(* Logix 5000 project; controller Sucrose_Main Emulate 5570 rev 20.12; software revision 20.01; part 24 of 30 *)
(* tags used below, declared in another part *)
   AI_E23_0 : REAL[8];   // Analog Input EN2T_FLX 192.168.1.23
   AI_E23_1 : REAL[8];   // Analog Input EN2T_FLX 192.168.1.23
   Alarm_ACK_Master_Timer : TIMER;
   CIPRemote : Area_Program;
   DI_E23_3 : ALIAS FOR FLX_E23:3:I;   // Discrete Input EN2T_FLX 192.168.1.23
   DI_E23_4 : ALIAS FOR FLX_E23:4:I;   // Discrete Input EN2T_FLX 192.168.1.23
   DI_E25_2 : ALIAS FOR FLX_E25:2:I;   // Discrete Input EN2T_FLX 192.168.1.25
   DO_E24_0 : ALIAS FOR FLX_E24:0:O;   // Discrete Output EN2T_FLX 192.168.1.24
   DO_E24_1 : ALIAS FOR FLX_E24:1:O;   // Discrete Output EN2T_FLX 192.168.1.24
   FV230006_AOI : QSI_Flow_Valve;   // FV-23-00-06 RETURN PIG TO LAUNCHER VALVE V7
   FV230007_AOI : QSI_Flow_Valve;   // FV-23-00-07 RETURN PIG TO LAUNCHER VALVE V6
   FV230101_AOI : QSI_Flow_Valve;   // FV-23-01-01-O SUCROSE RECEIVING TO SUCROSE TANK #1 VALVE OPEN
   FV230201_AOI : QSI_Flow_Valve;   // FV-23-02-01-O SUCROSE RECEIVING TO SUCROSE TANK #2 VALVE OPEN
   FV230301_AOI : QSI_Flow_Valve;   // FV-23-03-01-O SUCROSE RECEIVING TO SUCROSE TANK #3 VALVE OPEN
   ONESHOTBITS : INT[10];
   Rung_Comment : BOOL;
   Sucrose_MM_Enable : BOOL;
   SucroseCIP_RECEIVING_REMOTE : CIP_REMOTE;
   SucroseCIP_TK230101_REMOTE : CIP_REMOTE;
   SucroseCIP_TK230201_REMOTE : CIP_REMOTE;
   SucroseCIP_TK230301_REMOTE : CIP_REMOTE;
   SucroseReceiving : Area_Program;
   SucroseTanks : Area_Program;
   TK_23_01_01_HIGH_LEVEL : DINT;
   TK_23_01_01_RECEIVING_COMPLETE : BOOL;
   TK_23_02_01_HIGH_LEVEL : DINT;
   TK_23_02_01_RECEIVING_COMPLETE : BOOL;
   TK_23_03_01_HIGH_LEVEL : DINT;
   TK_23_03_01_RECEIVING_COMPLETE : BOOL;
(* ReceivingArea_AutoLogic, continued *)

ROUTINE Enable_Logic   (* ladder *)
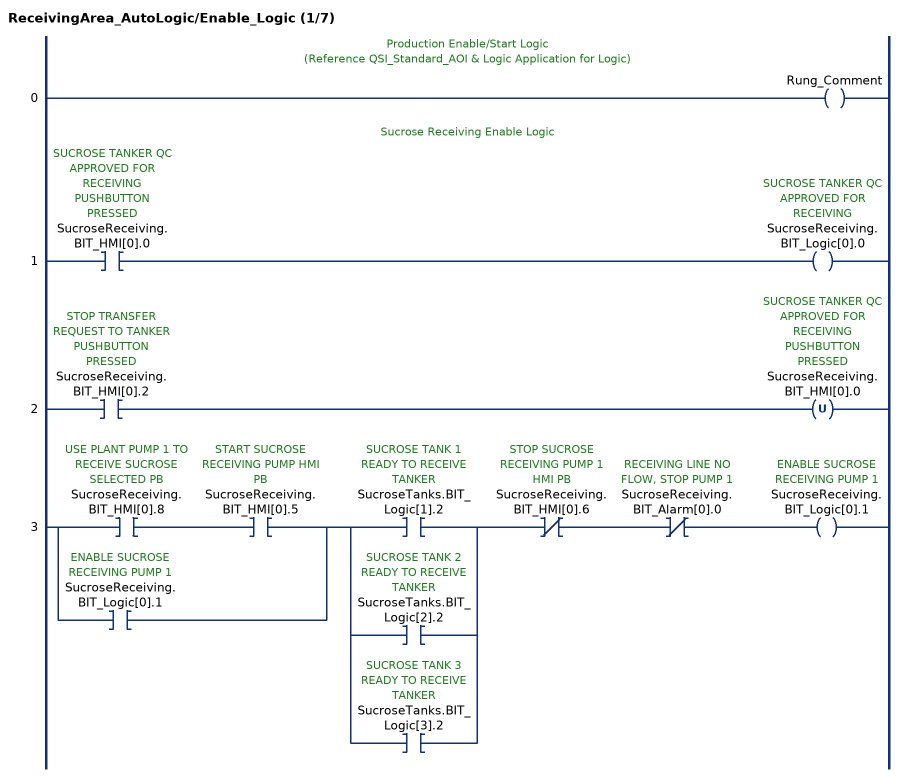
   // Production Enable/Start Logic
   // (Reference QSI_Standard_AOI & Logic Application for Logic)
   0: OTE(Rung_Comment);
   // Sucrose Receiving Enable Logic
   1: XIC(SucroseReceiving.BIT_HMI[0].0)OTE(SucroseReceiving.BIT_Logic[0].0);
   2: XIC(SucroseReceiving.BIT_HMI[0].2)OTU(SucroseReceiving.BIT_HMI[0].0);
   3: [XIC(SucroseReceiving.BIT_HMI[0].8) XIC(SucroseReceiving.BIT_HMI[0].5) ,XIC(SucroseReceiving.BIT_Logic[0].1) ][XIC(SucroseTanks.BIT_Logic[1].2) ,XIC(SucroseTanks.BIT_Logic[2].2) ,XIC(SucroseTanks.BIT_Logic[3].2) ]XIO(SucroseReceiving.BIT_HMI[0].6)XIO(SucroseReceiving.BIT_Alarm[0].0)OTE(SucroseReceiving.BIT_Logic[0].1);
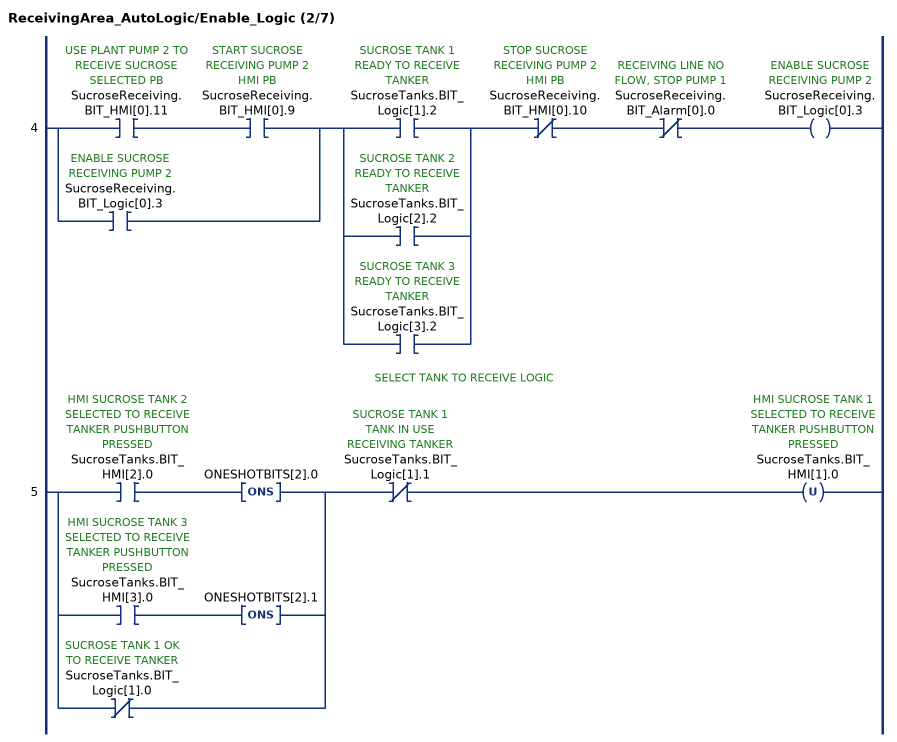
   4: [XIC(SucroseReceiving.BIT_HMI[0].11) XIC(SucroseReceiving.BIT_HMI[0].9) ,XIC(SucroseReceiving.BIT_Logic[0].3) ][XIC(SucroseTanks.BIT_Logic[1].2) ,XIC(SucroseTanks.BIT_Logic[2].2) ,XIC(SucroseTanks.BIT_Logic[3].2) ]XIO(SucroseReceiving.BIT_HMI[0].10)XIO(SucroseReceiving.BIT_Alarm[0].0)OTE(SucroseReceiving.BIT_Logic[0].3);
   // SELECT TANK TO RECEIVE LOGIC
   5: [XIC(SucroseTanks.BIT_HMI[2].0) ONS(ONESHOTBITS[2].0) ,XIC(SucroseTanks.BIT_HMI[3].0) ONS(ONESHOTBITS[2].1) ,XIO(SucroseTanks.BIT_Logic[1].0) ]XIO(SucroseTanks.BIT_Logic[1].1)OTU(SucroseTanks.BIT_HMI[1].0);
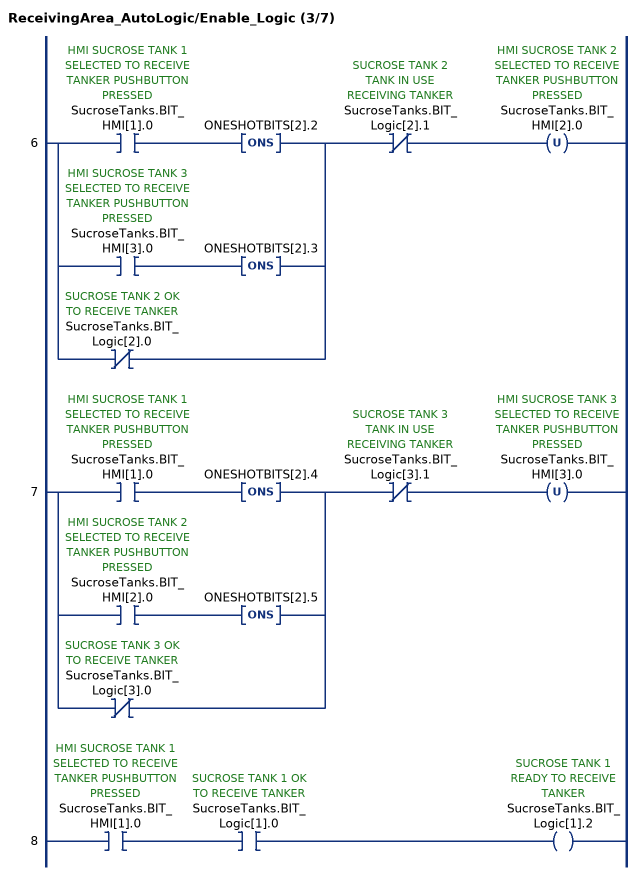
   6: [XIC(SucroseTanks.BIT_HMI[1].0) ONS(ONESHOTBITS[2].2) ,XIC(SucroseTanks.BIT_HMI[3].0) ONS(ONESHOTBITS[2].3) ,XIO(SucroseTanks.BIT_Logic[2].0) ]XIO(SucroseTanks.BIT_Logic[2].1)OTU(SucroseTanks.BIT_HMI[2].0);
   7: [XIC(SucroseTanks.BIT_HMI[1].0) ONS(ONESHOTBITS[2].4) ,XIC(SucroseTanks.BIT_HMI[2].0) ONS(ONESHOTBITS[2].5) ,XIO(SucroseTanks.BIT_Logic[3].0) ]XIO(SucroseTanks.BIT_Logic[3].1)OTU(SucroseTanks.BIT_HMI[3].0);
   8: XIC(SucroseTanks.BIT_HMI[1].0)XIC(SucroseTanks.BIT_Logic[1].0)OTE(SucroseTanks.BIT_Logic[1].2);
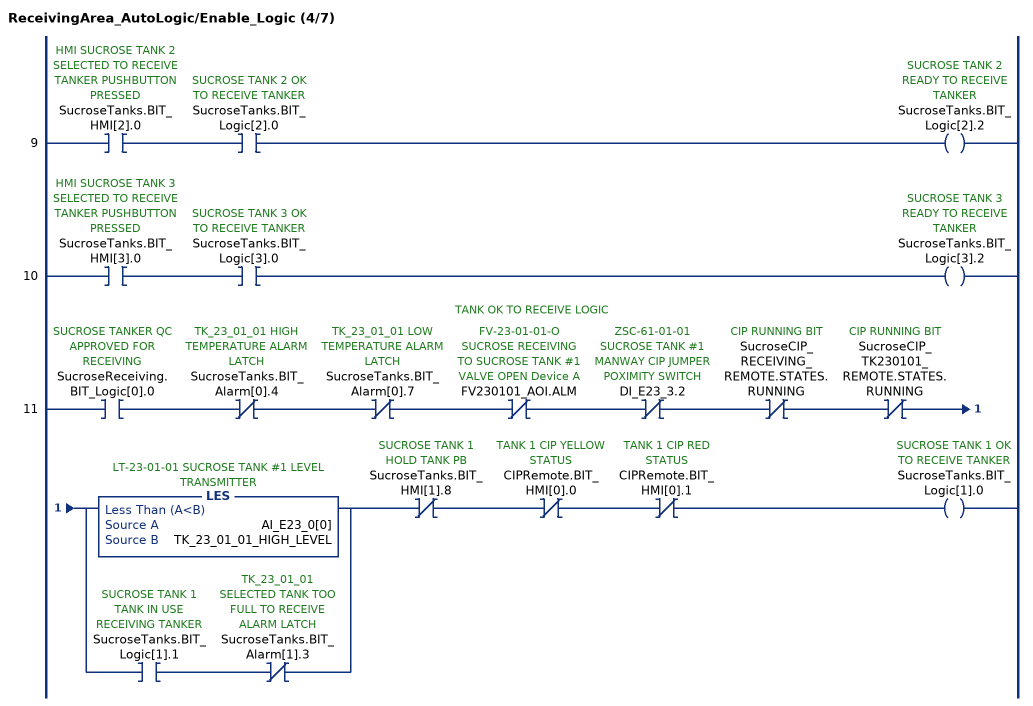
   9: XIC(SucroseTanks.BIT_HMI[2].0)XIC(SucroseTanks.BIT_Logic[2].0)OTE(SucroseTanks.BIT_Logic[2].2);
   10: XIC(SucroseTanks.BIT_HMI[3].0)XIC(SucroseTanks.BIT_Logic[3].0)OTE(SucroseTanks.BIT_Logic[3].2);
   // TANK OK TO RECEIVE LOGIC
   11: XIC(SucroseReceiving.BIT_Logic[0].0)XIO(SucroseTanks.BIT_Alarm[0].4)XIO(SucroseTanks.BIT_Alarm[0].7)XIO(FV230101_AOI.ALM)XIO(DI_E23_3.2)XIO(SucroseCIP_RECEIVING_REMOTE.STATES.RUNNING)XIO(SucroseCIP_TK230101_REMOTE.STATES.RUNNING)[LES(AI_E23_0[0],TK_23_01_01_HIGH_LEVEL) ,XIC(SucroseTanks.BIT_Logic[1].1) XIO(SucroseTanks.BIT_Alarm[1].3) ]XIO(SucroseTanks.BIT_HMI[1].8)XIO(CIPRemote.BIT_HMI[0].0)XIO(CIPRemote.BIT_HMI[0].1)OTE(SucroseTanks.BIT_Logic[1].0);
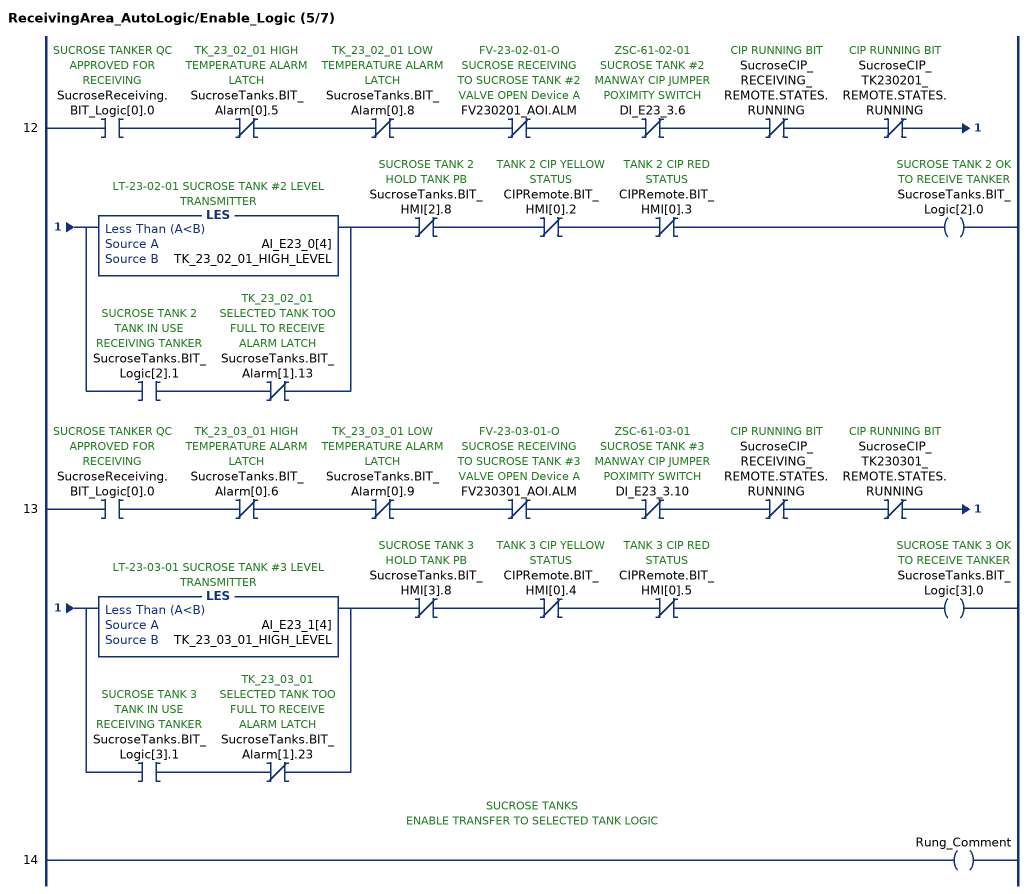
   12: XIC(SucroseReceiving.BIT_Logic[0].0)XIO(SucroseTanks.BIT_Alarm[0].5)XIO(SucroseTanks.BIT_Alarm[0].8)XIO(FV230201_AOI.ALM)XIO(DI_E23_3.6)XIO(SucroseCIP_RECEIVING_REMOTE.STATES.RUNNING)XIO(SucroseCIP_TK230201_REMOTE.STATES.RUNNING)[LES(AI_E23_0[4],TK_23_02_01_HIGH_LEVEL) ,XIC(SucroseTanks.BIT_Logic[2].1) XIO(SucroseTanks.BIT_Alarm[1].13) ]XIO(SucroseTanks.BIT_HMI[2].8)XIO(CIPRemote.BIT_HMI[0].2)XIO(CIPRemote.BIT_HMI[0].3)OTE(SucroseTanks.BIT_Logic[2].0);
   13: XIC(SucroseReceiving.BIT_Logic[0].0)XIO(SucroseTanks.BIT_Alarm[0].6)XIO(SucroseTanks.BIT_Alarm[0].9)XIO(FV230301_AOI.ALM)XIO(DI_E23_3.10)XIO(SucroseCIP_RECEIVING_REMOTE.STATES.RUNNING)XIO(SucroseCIP_TK230301_REMOTE.STATES.RUNNING)[LES(AI_E23_1[4],TK_23_03_01_HIGH_LEVEL) ,XIC(SucroseTanks.BIT_Logic[3].1) XIO(SucroseTanks.BIT_Alarm[1].23) ]XIO(SucroseTanks.BIT_HMI[3].8)XIO(CIPRemote.BIT_HMI[0].4)XIO(CIPRemote.BIT_HMI[0].5)OTE(SucroseTanks.BIT_Logic[3].0);
   // SUCROSE TANKS
   // ENABLE TRANSFER TO SELECTED TANK LOGIC
   14: OTE(Rung_Comment);
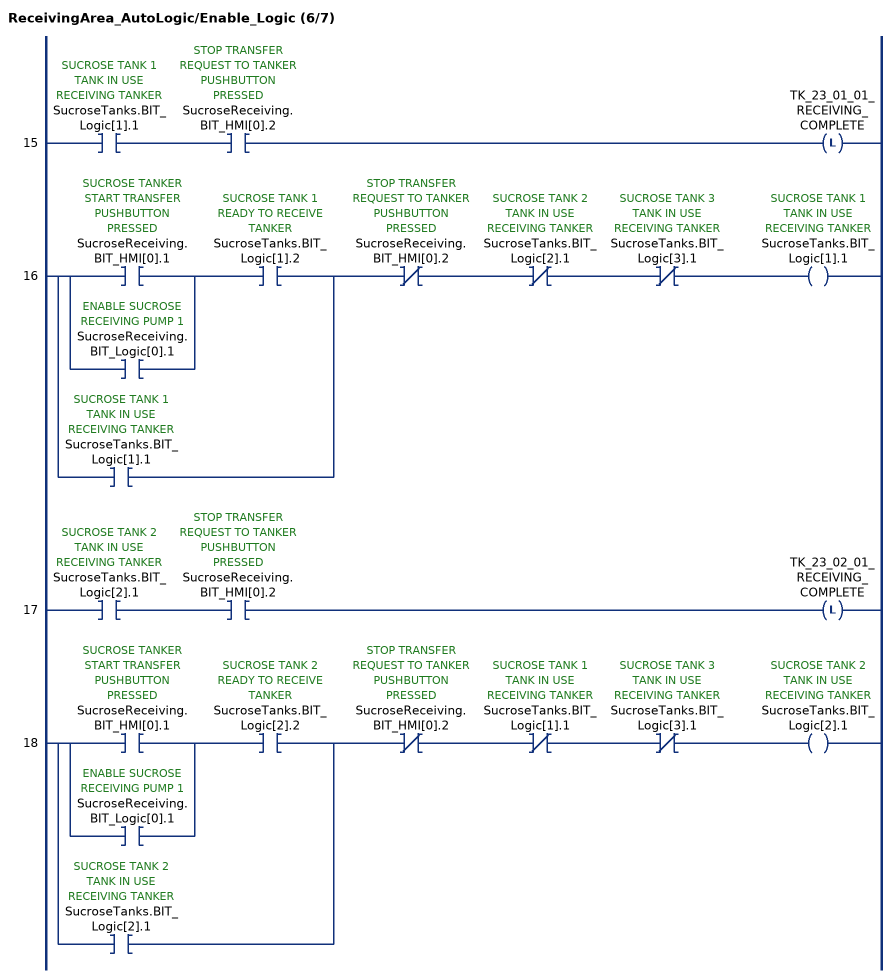
   15: XIC(SucroseTanks.BIT_Logic[1].1)XIC(SucroseReceiving.BIT_HMI[0].2)OTL(TK_23_01_01_RECEIVING_COMPLETE);
   16: [[XIC(SucroseReceiving.BIT_HMI[0].1) ,XIC(SucroseReceiving.BIT_Logic[0].1) ] XIC(SucroseTanks.BIT_Logic[1].2) ,XIC(SucroseTanks.BIT_Logic[1].1) ]XIO(SucroseReceiving.BIT_HMI[0].2)XIO(SucroseTanks.BIT_Logic[2].1)XIO(SucroseTanks.BIT_Logic[3].1)OTE(SucroseTanks.BIT_Logic[1].1);
   17: XIC(SucroseTanks.BIT_Logic[2].1)XIC(SucroseReceiving.BIT_HMI[0].2)OTL(TK_23_02_01_RECEIVING_COMPLETE);
   18: [[XIC(SucroseReceiving.BIT_HMI[0].1) ,XIC(SucroseReceiving.BIT_Logic[0].1) ] XIC(SucroseTanks.BIT_Logic[2].2) ,XIC(SucroseTanks.BIT_Logic[2].1) ]XIO(SucroseReceiving.BIT_HMI[0].2)XIO(SucroseTanks.BIT_Logic[1].1)XIO(SucroseTanks.BIT_Logic[3].1)OTE(SucroseTanks.BIT_Logic[2].1);
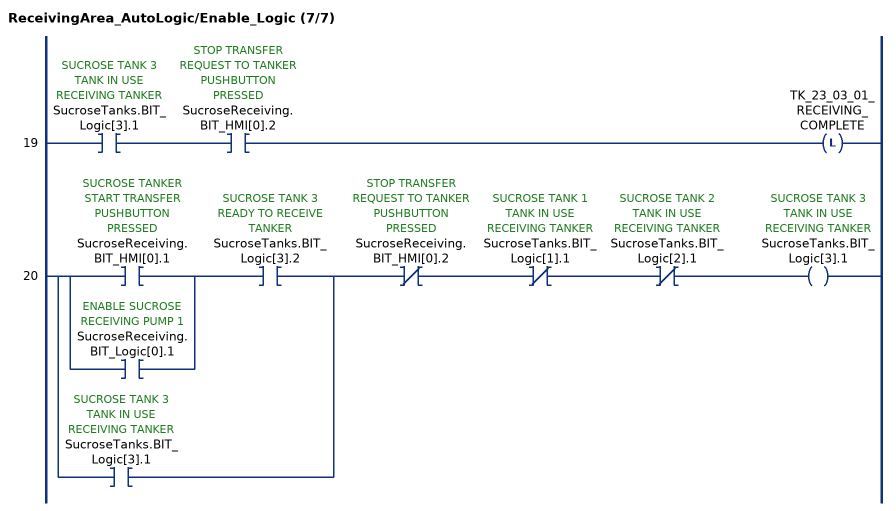
   19: XIC(SucroseTanks.BIT_Logic[3].1)XIC(SucroseReceiving.BIT_HMI[0].2)OTL(TK_23_03_01_RECEIVING_COMPLETE);
   20: [[XIC(SucroseReceiving.BIT_HMI[0].1) ,XIC(SucroseReceiving.BIT_Logic[0].1) ] XIC(SucroseTanks.BIT_Logic[3].2) ,XIC(SucroseTanks.BIT_Logic[3].1) ]XIO(SucroseReceiving.BIT_HMI[0].2)XIO(SucroseTanks.BIT_Logic[1].1)XIO(SucroseTanks.BIT_Logic[2].1)OTE(SucroseTanks.BIT_Logic[3].1);
END_ROUTINE

ROUTINE MainRoutine   (* ladder *)
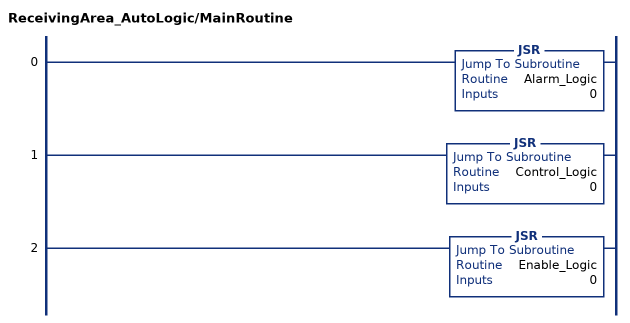
   0: JSR(Alarm_Logic,0);
   1: JSR(Control_Logic,0);
   2: JSR(Enable_Logic,0);
END_ROUTINE
END_PROGRAM

PROGRAM ReceivingArea_EN2T_IO_Discrete_DO_E24_0   (* main routine MainRoutine *)

ROUTINE _00_FV230006   (* ladder *)
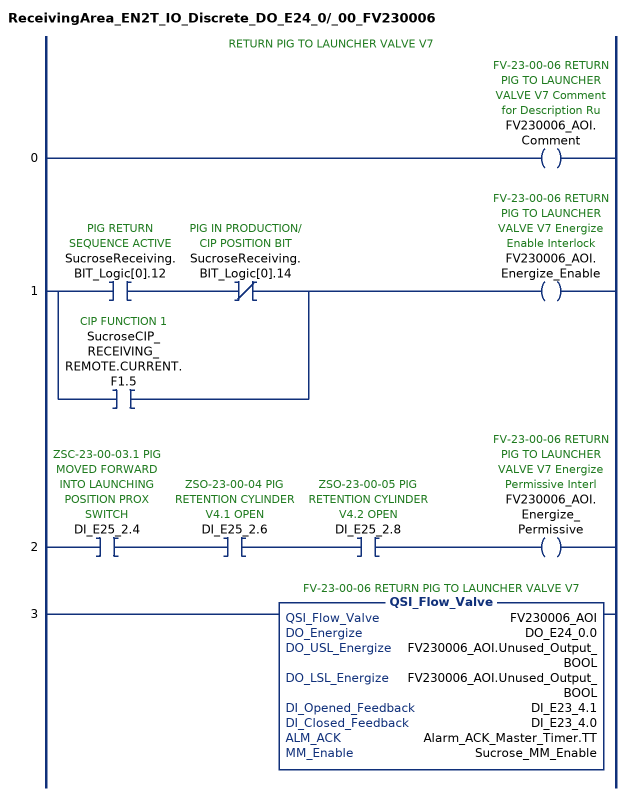
   // RETURN PIG TO LAUNCHER VALVE V7
   0: OTE(FV230006_AOI.Comment);
   1: [XIC(SucroseReceiving.BIT_Logic[0].12) XIO(SucroseReceiving.BIT_Logic[0].14) ,XIC(SucroseCIP_RECEIVING_REMOTE.CURRENT.F1.5) ]OTE(FV230006_AOI.Energize_Enable);
   2: XIC(DI_E25_2.4)XIC(DI_E25_2.6)XIC(DI_E25_2.8)OTE(FV230006_AOI.Energize_Permissive);
   3: QSI_Flow_Valve(FV230006_AOI,DO_E24_0.0,FV230006_AOI.Unused_Output_BOOL,FV230006_AOI.Unused_Output_BOOL,DI_E23_4.1,DI_E23_4.0,Alarm_ACK_Master_Timer.TT,Sucrose_MM_Enable);
END_ROUTINE

ROUTINE _01_FV230007   (* ladder *)
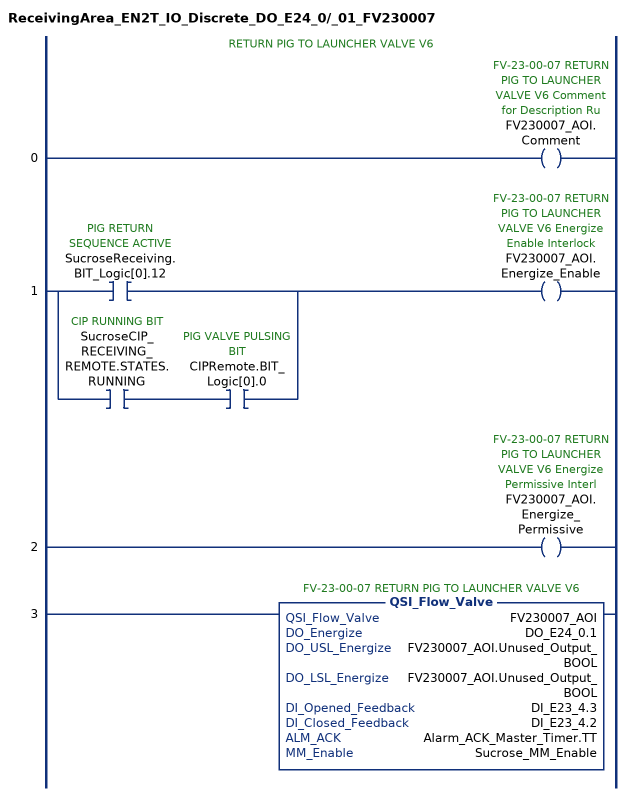
   // RETURN PIG TO LAUNCHER VALVE V6
   0: OTE(FV230007_AOI.Comment);
   1: [XIC(SucroseReceiving.BIT_Logic[0].12) ,XIC(SucroseCIP_RECEIVING_REMOTE.STATES.RUNNING) XIC(CIPRemote.BIT_Logic[0].0) ]OTE(FV230007_AOI.Energize_Enable);
   2: OTE(FV230007_AOI.Energize_Permissive);
   3: QSI_Flow_Valve(FV230007_AOI,DO_E24_0.1,FV230007_AOI.Unused_Output_BOOL,FV230007_AOI.Unused_Output_BOOL,DI_E23_4.3,DI_E23_4.2,Alarm_ACK_Master_Timer.TT,Sucrose_MM_Enable);
END_ROUTINE

ROUTINE _02_FV230101   (* ladder *)
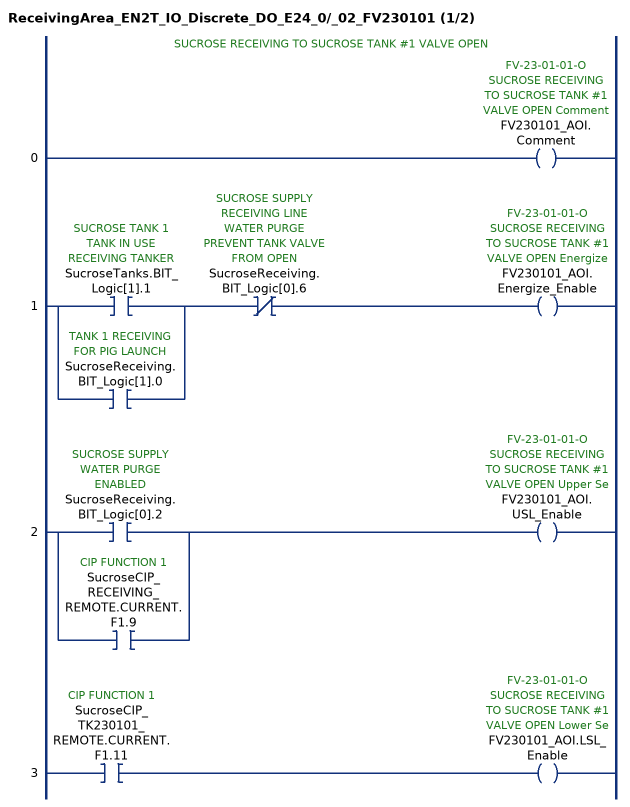
   // SUCROSE RECEIVING TO SUCROSE TANK #1 VALVE OPEN
   0: OTE(FV230101_AOI.Comment);
   1: [XIC(SucroseTanks.BIT_Logic[1].1) ,XIC(SucroseReceiving.BIT_Logic[1].0) ]XIO(SucroseReceiving.BIT_Logic[0].6)OTE(FV230101_AOI.Energize_Enable);
   2: [XIC(SucroseReceiving.BIT_Logic[0].2) ,XIC(SucroseCIP_RECEIVING_REMOTE.CURRENT.F1.9) ]OTE(FV230101_AOI.USL_Enable);
   3: XIC(SucroseCIP_TK230101_REMOTE.CURRENT.F1.11)OTE(FV230101_AOI.LSL_Enable);
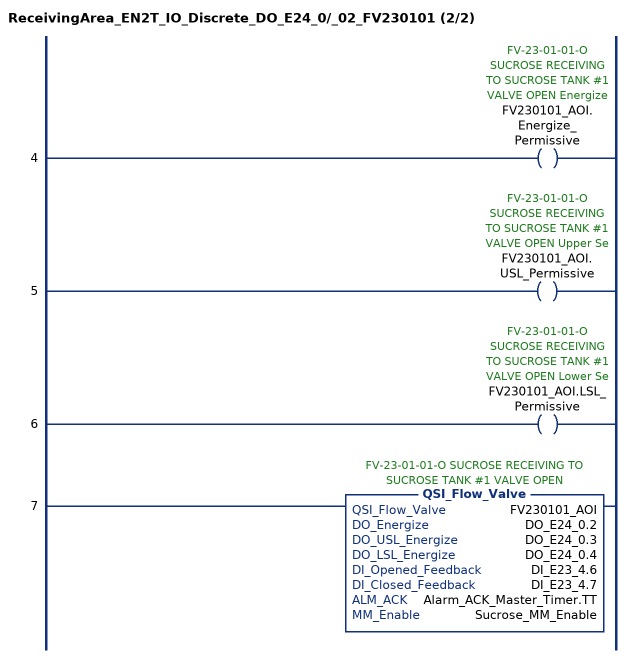
   4: OTE(FV230101_AOI.Energize_Permissive);
   5: OTE(FV230101_AOI.USL_Permissive);
   6: OTE(FV230101_AOI.LSL_Permissive);
   7: QSI_Flow_Valve(FV230101_AOI,DO_E24_0.2,DO_E24_0.3,DO_E24_0.4,DI_E23_4.6,DI_E23_4.7,Alarm_ACK_Master_Timer.TT,Sucrose_MM_Enable);
END_ROUTINE

ROUTINE _08_FV230201   (* ladder *)
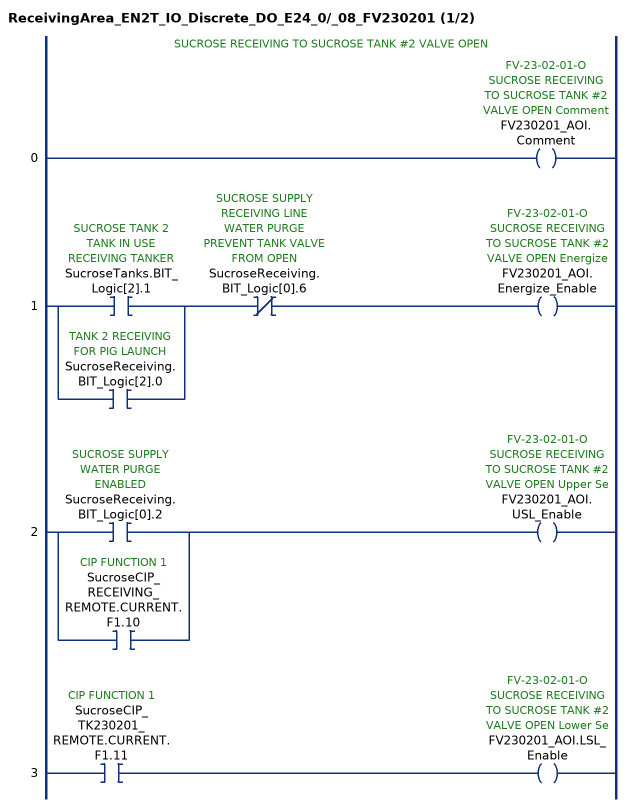
   // SUCROSE RECEIVING TO SUCROSE TANK #2 VALVE OPEN
   0: OTE(FV230201_AOI.Comment);
   1: [XIC(SucroseTanks.BIT_Logic[2].1) ,XIC(SucroseReceiving.BIT_Logic[2].0) ]XIO(SucroseReceiving.BIT_Logic[0].6)OTE(FV230201_AOI.Energize_Enable);
   2: [XIC(SucroseReceiving.BIT_Logic[0].2) ,XIC(SucroseCIP_RECEIVING_REMOTE.CURRENT.F1.10) ]OTE(FV230201_AOI.USL_Enable);
   3: XIC(SucroseCIP_TK230201_REMOTE.CURRENT.F1.11)OTE(FV230201_AOI.LSL_Enable);
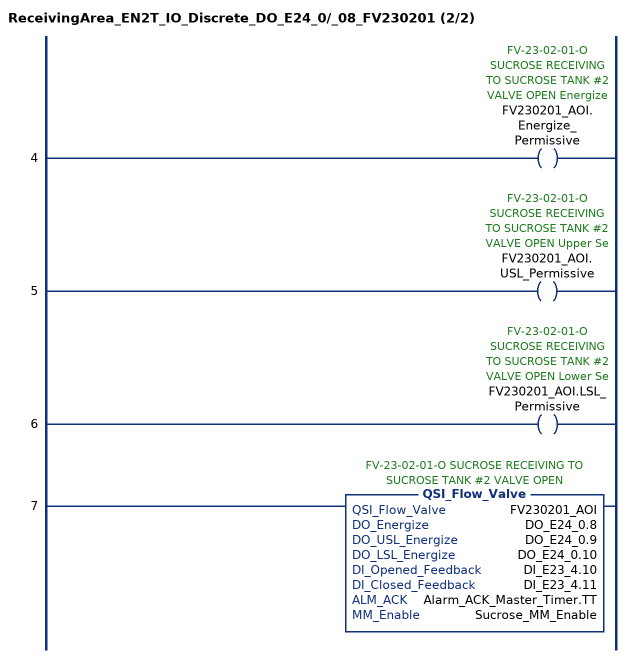
   4: OTE(FV230201_AOI.Energize_Permissive);
   5: OTE(FV230201_AOI.USL_Permissive);
   6: OTE(FV230201_AOI.LSL_Permissive);
   7: QSI_Flow_Valve(FV230201_AOI,DO_E24_0.8,DO_E24_0.9,DO_E24_0.10,DI_E23_4.10,DI_E23_4.11,Alarm_ACK_Master_Timer.TT,Sucrose_MM_Enable);
END_ROUTINE

ROUTINE MainRoutine   (* ladder *)
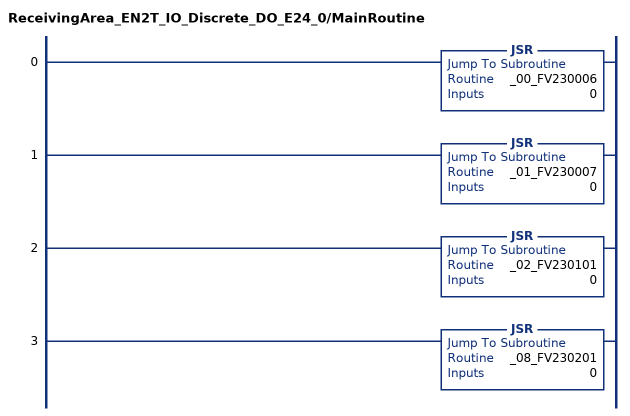
   0: JSR(_00_FV230006,0);
   1: JSR(_01_FV230007,0);
   2: JSR(_02_FV230101,0);
   3: JSR(_08_FV230201,0);
END_ROUTINE
END_PROGRAM

PROGRAM ReceivingArea_EN2T_IO_Discrete_DO_E24_1   (* main routine MainRoutine *)

ROUTINE _00_FV230301   (* ladder *)
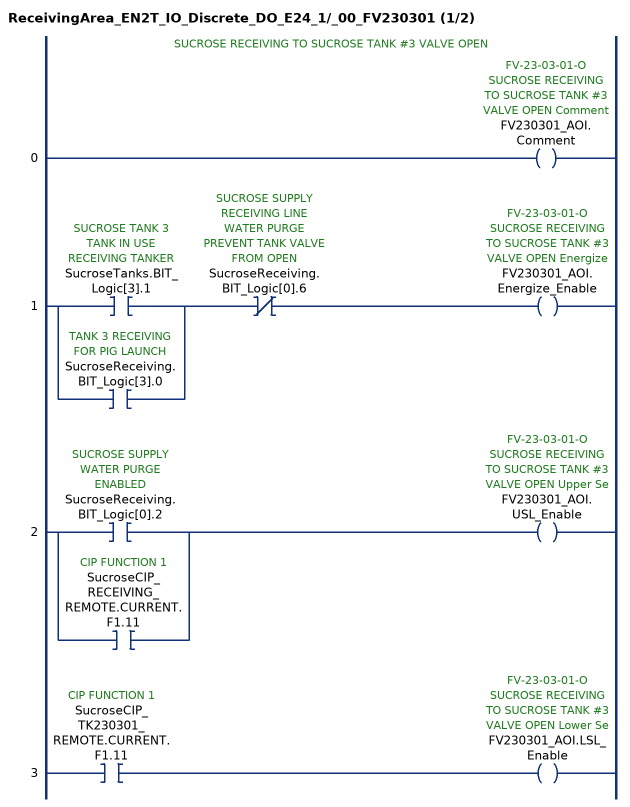
   // SUCROSE RECEIVING TO SUCROSE TANK #3 VALVE OPEN
   0: OTE(FV230301_AOI.Comment);
   1: [XIC(SucroseTanks.BIT_Logic[3].1) ,XIC(SucroseReceiving.BIT_Logic[3].0) ]XIO(SucroseReceiving.BIT_Logic[0].6)OTE(FV230301_AOI.Energize_Enable);
   2: [XIC(SucroseReceiving.BIT_Logic[0].2) ,XIC(SucroseCIP_RECEIVING_REMOTE.CURRENT.F1.11) ]OTE(FV230301_AOI.USL_Enable);
   3: XIC(SucroseCIP_TK230301_REMOTE.CURRENT.F1.11)OTE(FV230301_AOI.LSL_Enable);
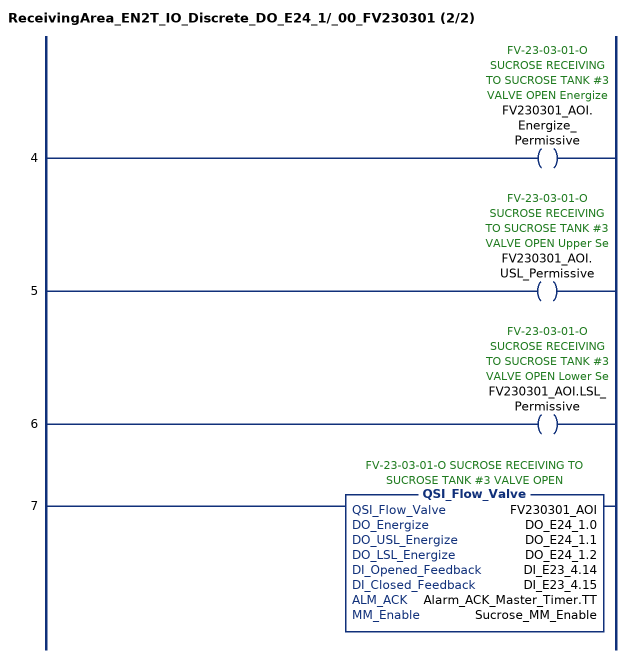
   4: OTE(FV230301_AOI.Energize_Permissive);
   5: OTE(FV230301_AOI.USL_Permissive);
   6: OTE(FV230301_AOI.LSL_Permissive);
   7: QSI_Flow_Valve(FV230301_AOI,DO_E24_1.0,DO_E24_1.1,DO_E24_1.2,DI_E23_4.14,DI_E23_4.15,Alarm_ACK_Master_Timer.TT,Sucrose_MM_Enable);
END_ROUTINE

ROUTINE MainRoutine   (* ladder *)
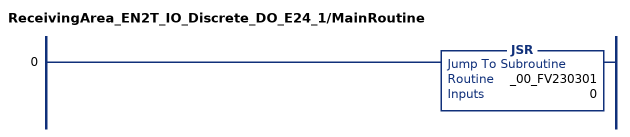
   0: JSR(_00_FV230301,0);
END_ROUTINE
END_PROGRAM
